FUNCTION_BLOCK ADD_VALUE_TO_VECTOR (* Adds a value to one of the vector components *)
  (* Standard: 61499-2 *)
  (* Version 1.0, 12-04-2012, GASR, Universidade do Estado de Santa Catarina *)
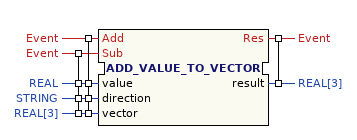
  EVENT_INPUT
    Add WITH value, direction, vector;
    Sub WITH value, direction, vector;
  END_EVENT
  EVENT_OUTPUT
    Res WITH result;
  END_EVENT
  VAR_INPUT
    value : REAL := 0; (* Value *)
    direction : STRING; (* x, y or z *)
    vector : ARRAY [0..2] OF REAL; (* Vector to do the operation *)
  END_VAR
  VAR_OUTPUT
    result : ARRAY [0..2] OF REAL;
  END_VAR
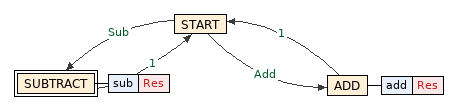
  EC_STATES
    SUBTRACT : sub -> Res;
    ADD : add -> Res;
    START;
  END_STATES
  EC_TRANSITIONS
    START TO ADD := Add;
    START TO SUBTRACT := Sub;
    ADD TO START := 1;
    SUBTRACT TO START := 1;
  END_TRANSITIONS
  ALGORITHM sub IN Lua:
 if( direction == 'x' ) then  result[1] = vector[1] - value  result[2] = vector[2]  result[3] = vector[3] elseif( direction == 'y' ) then  result[1] = vector[1]  result[2] = vector[2] - value  result[3] = vector[3] elseif( direction == 'z' ) then  result[1] = vector[1]  result[2] = vector[2]  result[3] = vector[3] - value  print( 'Subtratcing value', vector[1],vector[2],vector[3], 'value: '..value, result[1], result[2], result[3],direction ) end
  END_ALGORITHM
  ALGORITHM add IN Lua:
 if( direction == 'x' ) then  result[1] = vector[1] + value  result[2] = vector[2]  result[3] = vector[3] elseif( direction == 'y' ) then  result[1] = vector[1]  result[2] = vector[2] + value  result[3] = vector[3] elseif( direction == 'z' ) then  result[1] = vector[1]  result[2] = vector[2]  result[3] = vector[3] + value end
  END_ALGORITHM
END_FUNCTION_BLOCK
